{attribute addProperty BoxType "EP2316-0008-0016"}
{attribute addProperty Id "DO_InputsAT %I*DO_Inputs_9F71B9E27290DO_Diag_InputsAT %I*DO_Diag_Inputs_AC4A9AF06480DO_Inputs_DeviceAT %I*DO_Inputs_Device_BB3041553240DO_OutputsAT %Q*DO_Outputs_33B763766480DO_Outputs_DeviceAT %Q*DO_Outputs_Device_735003021620WcStateAT %I*WcState_F855686C1620InfoDataAT %I*InfoData_BC63D37F80100"}
{attribute addProperty CRC "1915324422"}
{attribute addProperty SizeInBites "344"}
{attribute addProperty SizeInBytes "43"}
TYPE EP2316_0F29F8B0 :
STRUCT
	{attribute addProperty Name "DO_Inputs"}
	DO_Inputs : DO_Inputs_9F71B9E2;
	{attribute addProperty Name "DO_Diag_Inputs"}
	DO_Diag_Inputs : DO_Diag_Inputs_AC4A9AF0;
	{attribute addProperty Name "DO_Inputs_Device"}
	DO_Inputs_Device : DO_Inputs_Device_BB304155;
	{attribute addProperty Name "DO_Outputs"}
	DO_Outputs : DO_Outputs_33B76376;
	{attribute addProperty Name "DO_Outputs_Device"}
	DO_Outputs_Device : DO_Outputs_Device_73500302;
	{attribute addProperty Name "WcState"}
	WcState : WcState_F855686C;
	{attribute addProperty Name "InfoData"}
	InfoData : InfoData_BC63D37F;
END_STRUCT
END_TYPE

(* stored: Version 1.2.0.0, ProductVersion 3.1.4024.9
   DUT EP2316_0F29F8B0: Id {1ec82755-4a10-4ed8-aab3-5161e5d733fe} *)
